# EPICS autosave request: iocBoot/obsolete/ioc13idd/auto_positions.req
file "CARS_80_motor_positions.req", P=$(P)
file "CARS_motor_positions.req", P=$(P), M=m85
file "CARS_motor_positions.req", P=$(P), M=m86
file "CARS_motor_positions.req", P=$(P), M=m87
file "CARS_motor_positions.req", P=$(P), M=m88
file "CARS_motor_positions.req", P=$(P), M=m89
file "CARS_motor_positions.req", P=$(P), M=m90
file "CARS_motor_positions.req", P=$(P), M=m91
file "CARS_motor_positions.req", P=$(P), M=m92
